(* PLC project Generated.project, CODESYS CODESYS V3.5 SP19 Patch 1 *)
(* stored: creationDateTime 2026-09-06T13:00:42.480247, modificationDateTime 2026-09-06T13:00:42.480247 *)

TYPE ST_ChainWinch : STRUCT
  Inputs_100 : ST_Chain_Winch_Inputs;
  Demandes_200 : ST_Chain_Winch_Demandes;
  Safety_300 : ST_Chain_Winch_Safety;
  Control_400 : ST_Chain_Winch_Control;
  Outputs_500 : ST_Chain_Winch_Outputs;
END_STRUCT;
END_TYPE

TYPE ST_Chain_Winch_Control : STRUCT
  Idx401_MotionAllowed : BOOL;  (* 1 = Prêt / Mouvement Autorisé | 0 = Bloqué *)
  Idx402_SpeedStepCalculated : INT;  (* Palier Vitesse Calculé (0, 1, 2, 3, 4) *)
  Idx403_SpeedRamp_Pct : REAL;  (* [%] Consigne Vitesse après Rampe *)
  Idx404_BrakeReleaseAuthorized : BOOL;  (* 1 = Ordre Ouverture Frein | 0 = Ordre Serrage *)
  Idx405_FinalInterlockState : E_WinchFinalInterlockState;  (* 🛡️ État frontière *)
  Idx406_FinalInterlockReason : E_WinchFinalInterlockReason;  (* 🛡️ Cause mémorisée *)
  Idx407_FinalAuthorizedStep : INT;  (* 🪜 Palier réellement autorisé *)
  Idx408_BrakeCommandOpenConfirmed : BOOL;  (* 🔌 Contacteur/bobine, pas frein mécanique *)
  Idx409_BrakeTimeoutElapsed : TIME;  (* ⏱️ Watchdog 500ms écoulé *)
  Idx410_RestartDelayElapsed : TIME;  (* ⏱️ Verrou 900ms écoulé *)
  Idx411_StepDelayElapsed : TIME;  (* ⏱️ Délai palier 1s250 écoulé *)
  Idx412_InTopSlowdownZone : BOOL;  (* 🐢 Palier plafonné à 1, approche limite haute *)
  Idx413_InBottomSlowdownZone : BOOL;  (* 🐢 Palier plafonné à 1, approche limite basse (câble ou légale) *)
  Idx414_BottomLimitActiveM : REAL;  (* : Limite basse active (m) — câble physique OU légale, la plus restrictive *)
  Idx415_MotorRequest : BOOL;  (* 🔎 Diagnostic anti-redémarrage — "commande active mais rien ne tourne" 1 = demande moteur active (palier>0 ET un seul sens) | 0 = pas de demande vue par la barrière *)
  Idx416_RestartRequired : BOOL;  (* 1 = purge anti-redémarrage armée, AuthorizedStep force a 0 tant que non purgee *)
  Idx417_RestartInhibit : BOOL;  (* 1 = verrou latché (frein non confirmé), exige Reset conscient — distinct de Idx416 *)
  Idx418_NeutralRequestSeen : BOOL;  (* 1 = passage au neutre observé pendant un RestartInhibit (réarmement en cours) *)
END_STRUCT;
END_TYPE

TYPE ST_Chain_Winch_Demandes : STRUCT
  Idx201_JoyRawPhysical_ANA : INT;  (* [pts] Bruts convertisseur (-2048 à +2048) *)
  Idx202_JoyScaledPhysical_Pct : REAL;  (* [%] Consigne Joystick (-100% à +100%) *)
  Idx203_HmiManualCmd_BtnAscent : BOOL;  (* 1 = Appui Bouton Ascending IHM | 0 = Relâché *)
  Idx204_HmiManualCmd_BtnDescent : BOOL;  (* 1 = Appui Bouton Descending IHM | 0 = Relâché *)
  Idx205_CycleAutoCmd_Pct : REAL;  (* [%] Consigne auto envoyée par le Cycle *)
  Idx206_ModeActive : E_Mode;  (* Mode courant (MANU_N1, AUTO_N1, MAINT_N2...) *)
  Idx207_BypassOperatorComm : BOOL;  (* 0 = Comm Normale OK | 1 = Bypass Réseau Actif ⚠️ *)
  Idx208_ArbitratedSpeed_Pct : REAL;  (* [%] Consigne finale retenue après arbitrage *)
  Idx209_ArbitratedDirection : INT;  (* +1 = Ascending | 0 = Neutre | -1 = Descending *)
  Idx210_CoupledUserRequestDirection : INT;  (* +1 = Ascending | 0 = Neutre | -1 = Descending *)
  Idx211_CoupledUserRequestActive : BOOL;  (* 1 = demande utilisateur couplée active *)
END_STRUCT;
END_TYPE

TYPE ST_Chain_Winch_Inputs : STRUCT
  Idx101_EncoderRawPos : DINT;  (* [Valeur brutes pts] Codeur connecté *)
  Idx102_CablePos_M : REAL;  (* [mètres] Position calculée du câble *)
  Idx103_ContactorsReleased_DI : BOOL;  (* 1 = OK (Tous contacteurs retombés à l'arrêt) | 0 = Contacteur collé *)
  Idx104_BrakeApplied : BOOL;  (* TRUE = frein SERRÉ (NOT BrakeFeedback — IHM garde le sens serré) *)
  Idx105_ThermalOk_DI : BOOL;  (* 1 = Température OK (Sain) | 0 = Surchauffe Moteur M1 *)
END_STRUCT;
END_TYPE

TYPE ST_Chain_Winch_Outputs : STRUCT
  Idx501_CmdRelayAscent_RQ : BOOL;  (* 1 = Relais Ascending ON | 0 = OFF *)
  Idx502_CmdRelayDescent_RQ : BOOL;  (* 1 = Relais Descending ON | 0 = OFF *)
  Idx503_CmdSpeedContactor1_DQ : BOOL;  (* 1 = Contacteur Vitesse 1 ON | 0 = OFF *)
  Idx504_CmdSpeedContactor4_DQ : BOOL;  (* 1 = Contacteur Vitesse 4 ON (Plein Gaz) | 0 = OFF *)
  Idx505_CmdBrakeRelease_RQ : BOOL;  (* 1 = Bobine Frein Alimentée (Ouvert) | 0 = Non Alimentée (Serré) *)
END_STRUCT;
END_TYPE

TYPE ST_Chain_Winch_Safety : STRUCT
  Idx301_EmergencyChainClosed : BOOL;  (* 1 = Boucle Urgence OK (Armé) | 0 = Arrêt d'Urgence Appuyé *)
  Idx302_SafeStopActive : BOOL;  (* 0 = Sain (Autorisé) | 1 = Arrêt Rapide Métier Actif *)
  Idx303_PowerCutOffActive : BOOL;  (* 0 = Puissance OK | 1 = Coupure Puissance Sécurité *)
  Idx304_TopSensorPhysical_DI : BOOL;  (* 1 = Capteur Haut Libre (Sain) | 0 = Butée Haute Atteinte *)
  Idx305_TopSensorBypassActive : BOOL;  (* 0 = Capteur Actif | 1 = Capteur Haut Shunté IHM ⚠️ *)
  Idx306_AscentPermitEffective : BOOL;  (* 1 = Ascending Autorisée | 0 = ASCENDING BLOQUÉE *)
  Idx307_SlackCablePhysical_DI : BOOL;  (* 1 = Câble Tendu (Sain) | 0 = Mou de Câble Détecté *)
  Idx308_SlackCableBypassActive : BOOL;  (* 0 = Capteur Actif | 1 = Mou de Câble Shunté IHM ⚠️ *)
  Idx309_DescendPermitEffective : BOOL;  (* 1 = Descending Autorisée | 0 = DESCENDING BLOQUÉE *)
  Idx310_ErrorOperatorComm : BOOL;  (* Défauts safety déchiffrés (bits ErrorId) — visibles individuellement à l'IHM bit0 Perte communication opérateur (joystick CAN / heartbeat IHM) *)
  Idx311_ErrorEncoder : BOOL;  (* bit1 Perte codeur de ce treuil *)
  Idx312_ErrorPhaseRotation : BOOL;  (* bit4 Mauvaise rotation de phases *)
  Idx313_ErrorMecaA : BOOL;  (* bit7 Mouvement non commandé / roue libre *)
  Idx314_ErrorMecaB : BOOL;  (* bit8 Absence confirmation arrêt sans commande *)
  Idx315_ErrorMecaC : BOOL;  (* bit9 Glissement M1 pendant cycle benne *)
  Idx316_ErrorMecaD : BOOL;  (* bit11 Non-arrêt sur capteur haut *)
  Idx317_ErrorMecaE : BOOL;  (* bit12/13 Écart synchro critique M1/M2 *)
  Idx318_ErrorBrakeThermal : BOOL;  (* bit10 Surchauffe thermique frein commun *)
  Idx319_ErrorOppositeDir : BOOL;  (* bit14 Sens réel opposé au sens commandé *)
  Idx320_ErrorNoMovement : BOOL;  (* bit15 Absence de mouvement malgré commande *)
  Idx321_CfgTopLimitM : REAL;  (* ⛔ Bloc "Pourquoi la montée ne s'arrête pas à la limite haute ?" — diagnostic ordonné (lecture maintenance) : config + position → butée atteinte → bypass actifs. 📐 Limite haute effective active (m) = CfgCableLimitAscent_M *)
  Idx322_CablePosM : REAL;  (* 📐 Position câble courante (m) *)
  Idx323_TopLimitReached : BOOL;  (* 1 = position >= limite haute (hors homing) | 0 = en dessous *)
  Idx324_AscentBlockedByTopLimit : BOOL;  (* 1 = montée réellement coupée par la butée logicielle (AscentPermit=0) | 0 = limitée non bloquante (bypass ?) *)
  Idx325_BypassTopLimitSoftware : BOOL;  (* ⚠️ 1 = butée logicielle shunétee IHM (individuel) *)
  Idx326_BypassTopLimitSoftCommun : BOOL;  (* ⚠️ 1 = butée logicielle shunétee (commun) *)
  Idx327_BypassTopLimitSwitch : BOOL;  (* ⚠️ 1 = capteur fin de course haut shuné IHM (individuel) *)
  Idx328_BypassTopLimitSwitchCommun : BOOL;  (* ⚠️ 1 = capteur fin de course haut shuné (commun) *)
  Idx329_BypassGlobal : BOOL;  (* ⚠️ 1 = bypass global treuil (individuel) *)
  Idx330_BypassGlobalCommun : BOOL;  (* ⚠️ 1 = bypass global (commun) *)
END_STRUCT;
END_TYPE

(* values of E_WinchFinalInterlockReason: NONE: Aucun blocage actif; BRAKE_COMMAND_NOT_CONFIRMED: Absence confirmation ouverture frein > 500ms; RESTART_INHIBITED: Inhibition redemarrage actif; SENSE_DROP_TIMEOUT: T_max §3bis depasse sans confirmation retombee (AC7) *)

{attribute 'qualified_only'}
{attribute 'strict'}
TYPE E_WinchFinalInterlockReason : (NONE := 0, BRAKE_COMMAND_NOT_CONFIRMED := 1, RESTART_INHIBITED := 2, SENSE_DROP_TIMEOUT := 3);
END_TYPE

(* values of E_WinchFinalInterlockState: DISABLED: Desactive / Hors service; READY: Pret / Etat nominal; WAIT_BRAKE_COMMAND_CONFIRMATION: Attente confirmation feedback frein; WAIT_STEP_DELAY: Temporisation changement de palier; WAIT_RESTART_DELAY: Temporisation anti-court-cycle redemarrage; FAULT: Etat de defaut; WAIT_SENSE_DROP_CONFIRM: Maintien §3bis du contacteur de sens (AC6/AC7) *)

{attribute 'qualified_only'}
{attribute 'strict'}
TYPE E_WinchFinalInterlockState : (DISABLED := 0, READY := 1, WAIT_BRAKE_COMMAND_CONFIRMATION := 2, WAIT_STEP_DELAY := 3, WAIT_RESTART_DELAY := 4, FAULT := 5, WAIT_SENSE_DROP_CONFIRM := 6);
END_TYPE

(* values of E_Mode: DISABLE: Mode Désactivé / Veille de sécurité (sorties bloquées); MAINT_N1: Manuel Niveau 1 : Pilotage unitaire avec toutes sécurités actives; MAINT_N2: Manuel Niveau 2 : Pilotage dégradé (droits étendus + bypasses autorisés); SEMI_AUTO: Mode Semi-Automatique (séquenceur automatique) *)

{attribute 'qualified_only'}
{attribute 'strict'}
TYPE E_Mode : (DISABLE := 0, MAINT_N1 := 1, MAINT_N2 := 2, SEMI_AUTO := 3);
END_TYPE
